// TIA Portal V15.1 export
// export: Created 2024-06-21T08:41:08.5073367Z, ExportSetting WithDefaults, DisplayName Totally Integrated Automation Portal, DisplayVersion V15.1 Update 5, DisplayName TIA Portal Openness, DisplayVersion V15.1 Update 5, DisplayName SINAMICS Startdrive Advanced, DisplayVersion V15.1, DisplayName G130, G150, S120, S150, SINAMICS MV, S210, DisplayVersion V15.1, DisplayName G110M, G120, G120C, G120D, G120P, DisplayVersion V15.1, DisplayName STEP 7 Professional, DisplayVersion V15.1 Update 5, DisplayName STEP 7 Safety, DisplayVersion V15.1, DisplayName WinCC Professional, DisplayVersion V15.1 Update 5, DisplayName SIMATIC Visualization Architect, DisplayVersion V15.1
FUNCTION "LGBRollerIAnim" : Void   // FC6609, FBD
TITLE = LIAnimDWord / LGBRollerIAnim
{ S7_Optimized_Access := 'TRUE' }
AUTHOR : VCC
FAMILY : Anim
NAME : SIAnim
VERSION : 0.1
// =============================================================================
// Handles the conversion from bits to one Word for simple icon Animation. 
// =============================================================================
// stored: AutoNumber false, IsIECCheckEnabled false, SetENOAutomatically False, UDAEnableTagReadback false
   VAR_INPUT
      I_SetPos : Bool;   // Set position / Set Position
      I_ResetPos : Bool;   // Reset position / Reset Position
      I_Active : Bool;   // Active
      I_Visible : Bool;   // ObjectVisible
      I_OutOfUse : Bool;   // Object out of use
      I_IntlkSetTrfIn : Bool;   // Interlock for Set direction / Interlock for Set direction transfer IN
      I_IntlkSetTrfOut : Bool;   // Interlock for Set direction / Interlock for Set direction transfer OUT
      I_IntlkResetTrfIn : Bool;   // Interlock for Reset direction / Interlock for Reset direction transfer IN
      I_IntlkResetTrfOut : Bool;   // Interlock for Reset direction / Interlock for Reset direction transfer OUT
      I_VisibleIntlkSetTrfIn : Bool;   // Interlock alarm for Set direction / Interlock Alarm for Set direction / Visible Interlock for Set direction transfer IN
      I_VisibleIntlkSetTrfOut : Bool;   // Interlock alarm for Set direction / Interlock Alarm for Set direction / Visible Interlock for Set direction transfer OUT
      I_VisibleIntlkResetTrfIn : Bool;   // Interlock alarm for Reset direction / Interlock Alarm for Reset direction / Visible Interlock for Reset direction transfer IN
      I_VisibleIntlkResetTrfOut : Bool;   // Interlock alarm for Reset direction / Interlock Alarm for Reset direction / Visible Interlock for Reset direction transfer OUT
      I_ManualMode : Bool;   // Manual mode / Manual Mode
      I_FncSelInHMI : Bool;   // Manual selection from HMI
      I_AlarmA : Bool;   // AlarmA
      I_AlarmB : Bool;   // AlarmB
      I_AlarmC : Bool;   // AlarmC
      I_AlarmD : Bool;   // AlarmD
      I_SafetyOk : Bool;   // Safety Ok / Safety OK
      I_MotionStopNOk : Bool;   // Safety Ok / Motion Stop OK
   END_VAR
   VAR_OUTPUT
      H_IAnim : DWord;   // Icon animation Word / Icon Animation
   END_VAR
BEGIN

REGION Network 1: Icon animation Word / **** 1 - Inputs **** Set position
   // Set Position
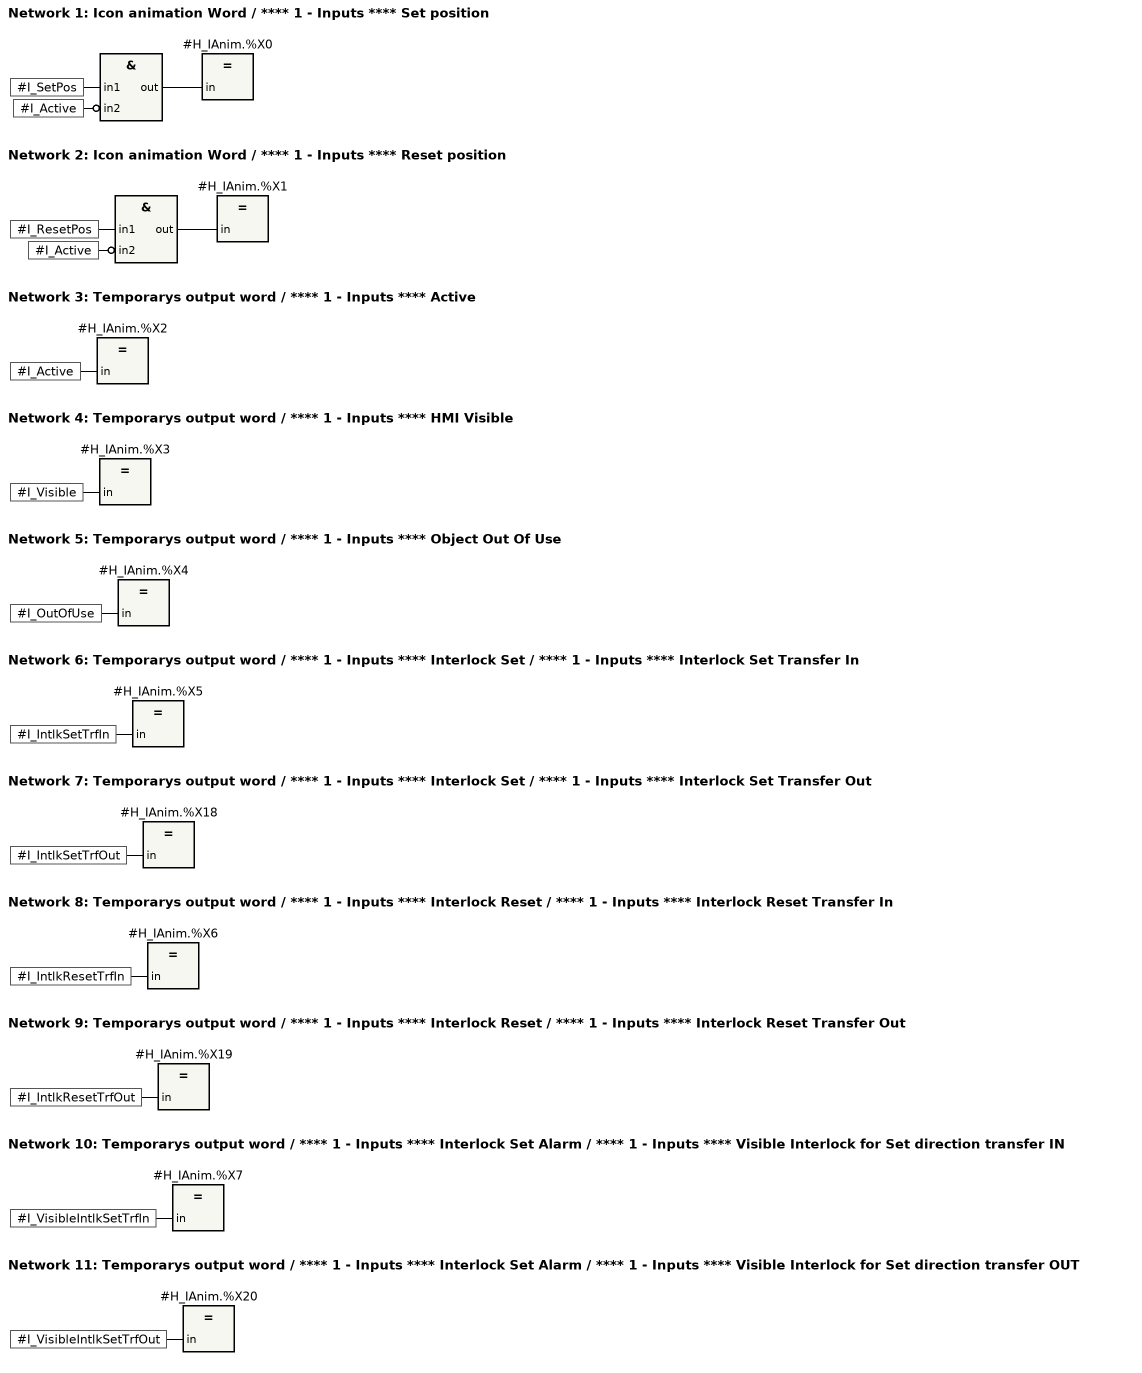
   #H_IAnim.%X0 := #I_SetPos AND NOT #I_Active;
END_REGION

REGION Network 2: Icon animation Word / **** 1 - Inputs **** Reset position
   // Reset Position
   #H_IAnim.%X1 := #I_ResetPos AND NOT #I_Active;
END_REGION

REGION Network 3: Temporarys output word / **** 1 - Inputs **** Active
   // Active
   #H_IAnim.%X2 := #I_Active;
END_REGION

REGION Network 4: Temporarys output word / **** 1 - Inputs **** HMI Visible
   // HMI Visible
   #H_IAnim.%X3 := #I_Visible;
END_REGION

REGION Network 5: Temporarys output word / **** 1 - Inputs **** Object Out Of Use
   // Object out of use
   #H_IAnim.%X4 := #I_OutOfUse;
END_REGION

REGION Network 6: Temporarys output word / **** 1 - Inputs **** Interlock Set / **** 1 - Inputs **** Interlock Set Transfer In
   // Interlock Set / Interlock Set Transfer In
   #H_IAnim.%X5 := #I_IntlkSetTrfIn;
END_REGION

REGION Network 7: Temporarys output word / **** 1 - Inputs **** Interlock Set / **** 1 - Inputs **** Interlock Set Transfer Out
   // Interlock Set / Interlock Set Transfer Out
   #H_IAnim.%X18 := #I_IntlkSetTrfOut;
END_REGION

REGION Network 8: Temporarys output word / **** 1 - Inputs **** Interlock Reset / **** 1 - Inputs **** Interlock Reset Transfer In
   // Interlock Reset / Interlock Reset Transfer In
   #H_IAnim.%X6 := #I_IntlkResetTrfIn;
END_REGION

REGION Network 9: Temporarys output word / **** 1 - Inputs **** Interlock Reset / **** 1 - Inputs **** Interlock Reset Transfer Out
   // Interlock Reset / Interlock Reset Transfer Out
   #H_IAnim.%X19 := #I_IntlkResetTrfOut;
END_REGION

REGION Network 10: Temporarys output word / **** 1 - Inputs **** Interlock Set Alarm / **** 1 - Inputs **** Visible Interlock for Set direction transfer IN
   // Interlock Set Alarm / Visible Interlock for Set direction transfer IN
   #H_IAnim.%X7 := #I_VisibleIntlkSetTrfIn;
END_REGION

REGION Network 11: Temporarys output word / **** 1 - Inputs **** Interlock Set Alarm / **** 1 - Inputs **** Visible Interlock for Set direction transfer OUT
   // Interlock Set Alarm / Visible Interlock for Set direction transfer OUT
   #H_IAnim.%X20 := #I_VisibleIntlkSetTrfOut;
END_REGION

REGION Network 12: Temporarys output word / **** 1 - Inputs **** Interlock Reset Alarm / **** 1 - Inputs **** Visible Interlock for Reset direction transfer IN
   // Interlock Reset Alarm / Visible Interlock for Reset direction transfer IN
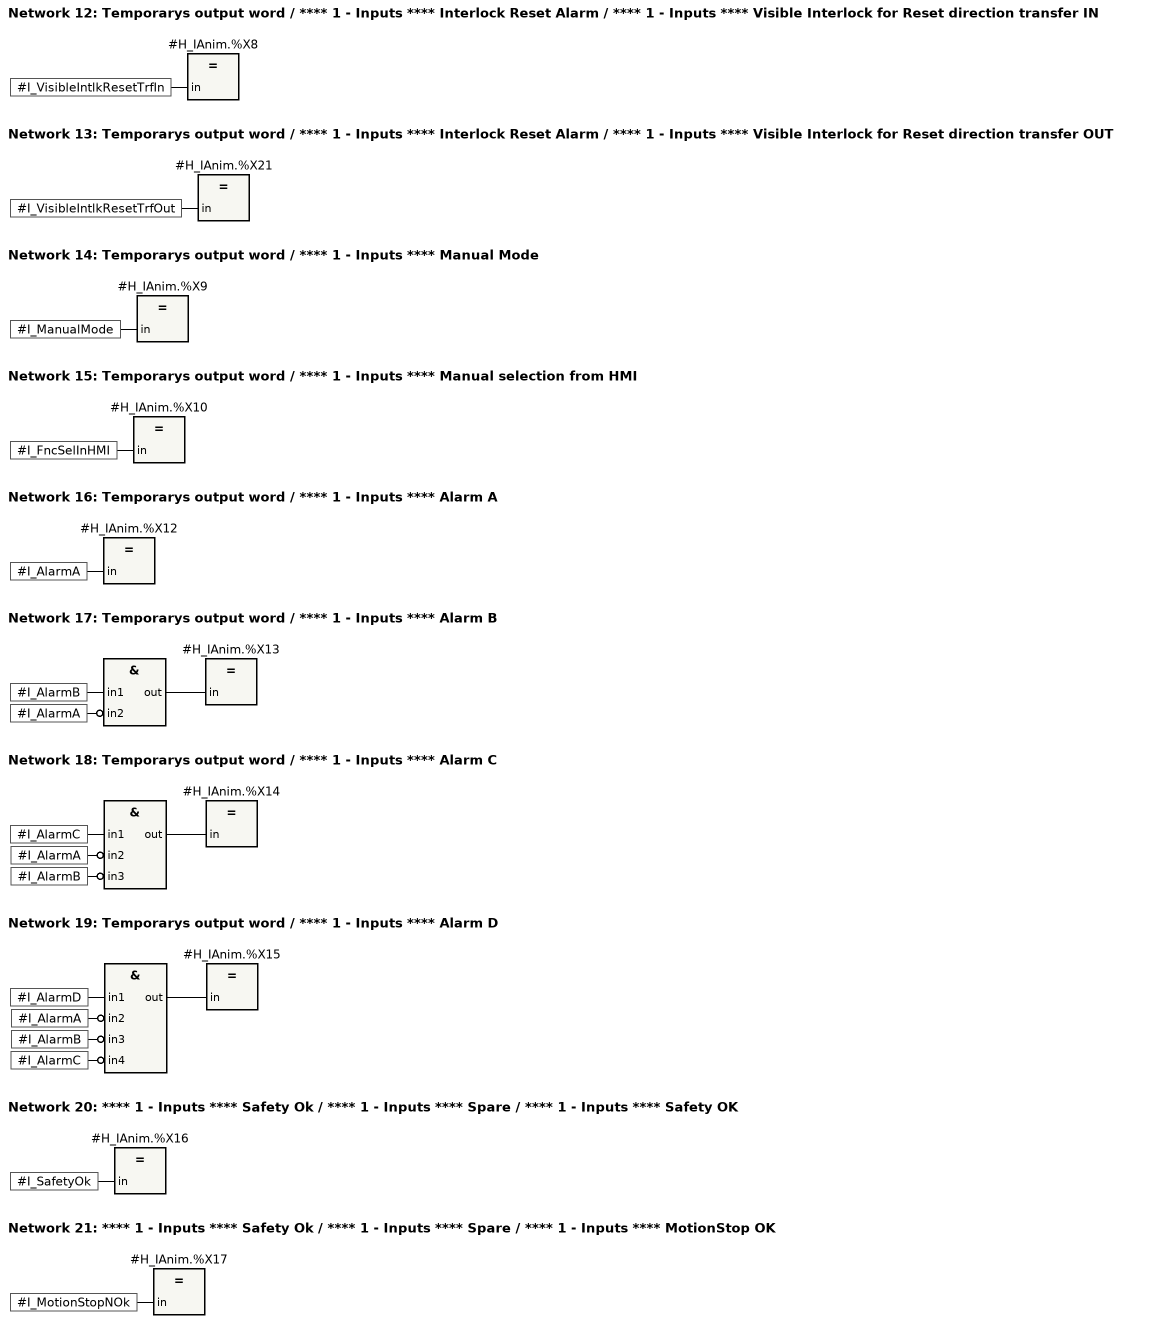
   #H_IAnim.%X8 := #I_VisibleIntlkResetTrfIn;
END_REGION

REGION Network 13: Temporarys output word / **** 1 - Inputs **** Interlock Reset Alarm / **** 1 - Inputs **** Visible Interlock for Reset direction transfer OUT
   // Interlock Reset Alarm / Visible Interlock for Reset direction transfer OUT
   #H_IAnim.%X21 := #I_VisibleIntlkResetTrfOut;
END_REGION

REGION Network 14: Temporarys output word / **** 1 - Inputs **** Manual Mode
   // Manual Mode
   #H_IAnim.%X9 := #I_ManualMode;
END_REGION

REGION Network 15: Temporarys output word / **** 1 - Inputs **** Manual selection from HMI
   // Manual selection from HMI
   #H_IAnim.%X10 := #I_FncSelInHMI;
END_REGION

REGION Network 16: Temporarys output word / **** 1 - Inputs **** Alarm A
   // Alarm A
   #H_IAnim.%X12 := #I_AlarmA;
END_REGION

REGION Network 17: Temporarys output word / **** 1 - Inputs **** Alarm B
   // Alarm B
   #H_IAnim.%X13 := #I_AlarmB AND NOT #I_AlarmA;
END_REGION

REGION Network 18: Temporarys output word / **** 1 - Inputs **** Alarm C
   // Alarm C
   #H_IAnim.%X14 := #I_AlarmC AND NOT #I_AlarmA AND NOT #I_AlarmB;
END_REGION

REGION Network 19: Temporarys output word / **** 1 - Inputs **** Alarm D
   // Alarm D
   #H_IAnim.%X15 := #I_AlarmD AND NOT #I_AlarmA AND NOT #I_AlarmB AND NOT #I_AlarmC;
END_REGION

REGION Network 20: **** 1 - Inputs **** Safety Ok / **** 1 - Inputs **** Spare / **** 1 - Inputs **** Safety OK
   // Safety Ok / Spare / Safety OK
   #H_IAnim.%X16 := #I_SafetyOk;
END_REGION

REGION Network 21: **** 1 - Inputs **** Safety Ok / **** 1 - Inputs **** Spare / **** 1 - Inputs **** MotionStop OK
   // Safety Ok / Spare / MotionStop OK
   #H_IAnim.%X17 := #I_MotionStopNOk;
END_REGION
END_FUNCTION
